FUNCTION "ST10_PartData" : Void
VAR_INPUT
  iSysMode : "RCS_SysComInterface_V1";
END_VAR
VAR_TEMP
  idex : Int;
END_VAR
BEGIN
  // Původní jazyk: SCL
  // Zdroj XML: EXPORT/Program blocks/OP010/12_PartData/ST10_PartData.xml
  // (Nebylo nalezeno StructuredText/FlgNet/StatementList; logika může být v GRAPH nebo v nepodporované reprezentaci.)
END_FUNCTION
